{attribute addProperty BoxType "EK1122-0000-0018"}
{attribute addProperty Id "Beckhoff_ELM35xxsub_EK1100EK1100_179A0949162"}
{attribute addProperty CRC "3090108780"}
{attribute addProperty SizeInBites "16"}
{attribute addProperty SizeInBytes "2"}
TYPE Beckhoff_ELM35xxEK1122_B82F516C EXTENDS EK1122_179A0949 :
STRUCT
	{attribute addProperty Name "Beckhoff_ELM35xxsub_EK1100"}
	Beckhoff_ELM35xxsub_EK1100 : EK1100_179A0949;
END_STRUCT
END_TYPE

(* stored: Version 1.2.0.0, ProductVersion 3.1.4024.9
   DUT Beckhoff_ELM35xxEK1122_B82F516C: Id {91050381-27ce-49af-9e07-9772d5fdaf09} *)
